{attribute 'qualified_only' := ''}
VAR_GLOBAL CONSTANT
    (*******************************************************************)
    (* Globale KONSTANTEN *)
    (*******************************************************************)

    USE_SIMULATION : BOOL := TRUE;

    STATION_NUMBER        : INT   := 18;
    MAX_GROUP             : INT   := 6;
    MAX_STATION_PER_GROUP : INT   := 8;
    MAX_RECIPE_NUMBER     : INT   := 4;
    MAX_TRACK_LENGTH      : LREAL := 10000;
    MAX_MOVER_SIZE        : LREAL := 200.0;
    MAX_VECTOR_LIST       : INT   := 10;

END_VAR

(* stored: Version 1.1.0.1, ProductVersion 3.1.4024.6
   GVL CONST: Id {9b3680ca-efd7-44b5-8e7f-6ff4b0673f03} *)
